SUBAPPLICATION Uebung_060_sub_Outputs (* für TC-SC also Task Controller Section Control *)
  (* Standard: 61499-2 *)
  (* Version 1.0, 2024-02-29, franz *)
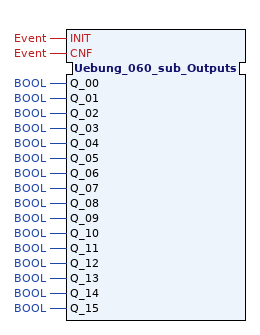
  EVENT_INPUT
    INIT;
    CNF;
  END_EVENT
  VAR_INPUT
    Q_00 : BOOL;
    Q_01 : BOOL;
    Q_02 : BOOL;
    Q_03 : BOOL;
    Q_04 : BOOL;
    Q_05 : BOOL;
    Q_06 : BOOL;
    Q_07 : BOOL;
    Q_08 : BOOL;
    Q_09 : BOOL;
    Q_10 : BOOL;
    Q_11 : BOOL;
    Q_12 : BOOL;
    Q_13 : BOOL;
    Q_14 : BOOL;
    Q_15 : BOOL;
  END_VAR
  FBS
    DigitalOutput_Q4 : QX(QI := TRUE);
    DigitalOutput_Q7 : QX(QI := TRUE);
    DigitalOutput_Q1 : QX(QI := TRUE);
    DigitalOutput_Q5 : QX(QI := TRUE);
    DigitalOutput_Q2 : QX(QI := TRUE);
    DigitalOutput_Q6 : QX(QI := TRUE);
    DigitalOutput_Q8 : QX(QI := TRUE);
    DigitalOutput_Q3 : QX(QI := TRUE);
    DigitalOutput_Q9 : QX(QI := TRUE);
    DigitalOutput_Q10 : QX(QI := TRUE);
    DigitalOutput_Q11 : QX(QI := TRUE);
    DigitalOutput_Q12 : QX(QI := TRUE);
    DigitalOutput_Q13 : QX(QI := TRUE);
    DigitalOutput_Q14 : QX(QI := TRUE);
    DigitalOutput_Q15 : QX(QI := TRUE);
    DigitalOutput_Q16 : QX(QI := TRUE);
  END_FBS
  EVENT_CONNECTIONS
    INIT TO DigitalOutput_Q4.INIT;
    CNF TO DigitalOutput_Q4.REQ;
    INIT TO DigitalOutput_Q7.INIT;
    CNF TO DigitalOutput_Q7.REQ;
    INIT TO DigitalOutput_Q1.INIT;
    CNF TO DigitalOutput_Q1.REQ;
    INIT TO DigitalOutput_Q5.INIT;
    CNF TO DigitalOutput_Q5.REQ;
    INIT TO DigitalOutput_Q2.INIT;
    CNF TO DigitalOutput_Q2.REQ;
    INIT TO DigitalOutput_Q6.INIT;
    CNF TO DigitalOutput_Q6.REQ;
    INIT TO DigitalOutput_Q8.INIT;
    CNF TO DigitalOutput_Q8.REQ;
    INIT TO DigitalOutput_Q3.INIT;
    CNF TO DigitalOutput_Q3.REQ;
    INIT TO DigitalOutput_Q9.INIT;
    CNF TO DigitalOutput_Q9.REQ;
    INIT TO DigitalOutput_Q10.INIT;
    CNF TO DigitalOutput_Q10.REQ;
    INIT TO DigitalOutput_Q11.INIT;
    CNF TO DigitalOutput_Q11.REQ;
    INIT TO DigitalOutput_Q12.INIT;
    CNF TO DigitalOutput_Q12.REQ;
    INIT TO DigitalOutput_Q13.INIT;
    CNF TO DigitalOutput_Q13.REQ;
    INIT TO DigitalOutput_Q14.INIT;
    CNF TO DigitalOutput_Q14.REQ;
    INIT TO DigitalOutput_Q15.INIT;
    CNF TO DigitalOutput_Q15.REQ;
    INIT TO DigitalOutput_Q16.INIT;
    CNF TO DigitalOutput_Q16.REQ;
  END_CONNECTIONS
  DATA_CONNECTIONS
    Q_06 TO DigitalOutput_Q7.OUT;
    Q_00 TO DigitalOutput_Q1.OUT;
    Q_04 TO DigitalOutput_Q5.OUT;
    Q_01 TO DigitalOutput_Q2.OUT;
    Q_05 TO DigitalOutput_Q6.OUT;
    Q_02 TO DigitalOutput_Q3.OUT;
    Q_03 TO DigitalOutput_Q4.OUT;
    Q_07 TO DigitalOutput_Q8.OUT;
    Q_08 TO DigitalOutput_Q9.OUT;
    Q_09 TO DigitalOutput_Q10.OUT;
    Q_10 TO DigitalOutput_Q11.OUT;
    Q_11 TO DigitalOutput_Q12.OUT;
    Q_12 TO DigitalOutput_Q13.OUT;
    Q_13 TO DigitalOutput_Q14.OUT;
    Q_14 TO DigitalOutput_Q15.OUT;
    Q_15 TO DigitalOutput_Q16.OUT;
  END_CONNECTIONS
END_SUBAPPLICATION
